PROGRAM MAIN
VAR
	eventEmitter_TestSuite : EventEmitter_TestSuite;
END_VAR

TcUnit.RUN();

END_PROGRAM

(* stored: Version 1.1.0.1, ProductVersion 3.1.4024.12
   POU MAIN: Id {0426f05b-5f97-0ad4-3f3a-5f3fc39bb59b}, SpecialFunc None *)
